// Core §3.8e(c) - where a mirror gets its owner's line data from. Pluggable
// like §3.8's recipe provider and §3.8b's store; the transport is a binding and
// deployment choice, and what it returns is untrusted input (§14).
INTERFACE I_LineSource

// Call every scan. TRUE on the scan a complete owner image was obtained.
METHOD M_Poll : BOOL
VAR_IN_OUT
    Image : ST_LineImage;
END_VAR
END_METHOD

// The last transport error, 0 when the last attempt succeeded.
METHOD M_Error : DINT
END_METHOD

END_INTERFACE

(* stored: Version 1.1.0.1, ProductVersion 3.1.4024.12
   Itf I_LineSource: Id {7737bb76-d8e3-4a3f-9299-cb43c60c8c92}
   Method M_Poll: Id {099847a0-f55e-448e-a765-4c62a2c41510}
   Method M_Error: Id {c93a877b-bfd1-4459-a789-882544d4c655} *)
